// TwinCAT 3 PLC project objectOriented
// ProgramVersion: 3.1.4024.0
// libraries:
//   Tc2_Standard, * (Beckhoff Automation GmbH)
//   Tc2_System, * (Beckhoff Automation GmbH)
//   Tc2_Utilities, * (Beckhoff Automation GmbH)
//   Tc3_Module, * (Beckhoff Automation GmbH)
// project tree:
//   DUTs/ E_EventType.TcDUT, ST_Event.TcDUT
//   / PlcTask.TcTTO
//   POUs/ EventLogger.TcPOU, FB_CsvlPersistentEventStorage.TcPOU, I_PersistentEventStorage.TcIO, MAIN.TcPOU, UpdateEventTimestampWithSystemTime.TcPOU

CONFIGURATION objectOriented
    RESOURCE PLC ON TwinCAT3
        TASK PlcTask(INTERVAL := T#10ms, PRIORITY := 21);
        PROGRAM MAIN WITH PlcTask : MAIN;
    END_RESOURCE
END_CONFIGURATION

// ---- DUTs/E_EventType.TcDUT
{attribute 'qualified_only'}
{attribute 'strict'}
{attribute 'to_string'}
TYPE E_EventType :
(
	Alarm := 0,
	Message := 1
);
END_TYPE

// ---- DUTs/ST_Event.TcDUT
TYPE ST_Event :
STRUCT
	eEventType : E_EventType;
	eEventSeverity : TcEventSeverity;
	nEventIdentity : UDINT;
	sEventText : STRING(255);
	dtTimeStamp : DATE_AND_TIME;
END_STRUCT
END_TYPE

// ---- POUs/I_PersistentEventStorage.TcIO
INTERFACE I_PersistentEventStorage

METHOD StoreEvent
VAR_INPUT
	stEvent : ST_Event;
END_VAR
END_METHOD

END_INTERFACE

// ---- POUs/MAIN.TcPOU
PROGRAM MAIN
VAR
//	UpdateEventTimestam : ST_Event;
	aBoolean : BOOL := FALSE;
		
	eEventType1 : E_EventType := E_EventType.Alarm;
	eEventSeverity1 : TcEventSeverity := TcEventSeverity.Error;
	nEventIdentity1 : UDINT := 42;
	sEventText1 : STRING(255) := 'This is a scary event';
	
	CsvPersistentEventStorage : FB_CsvlPersistentEventStorage;
	EventLogger : EventLogger(CsvPersistentEventStorage); // FB_init call leads to error
END_VAR

//IF NOT aBoolean THEN
//	UpdateEventTimestampWithSystemTime(stEvent := UpdateEventTimestam);
//	aBoolean := TRUE;
//END_IF

IF aBoolean THEN
	EventLogger.AddEvent(eEventType1, eEventSeverity1, nEventIdentity1, sEventText1);
	aBoolean := FALSE;
END_IF

CsvPersistentEventStorage();

END_PROGRAM

// ---- POUs/FB_CsvlPersistentEventStorage.TcPOU
FUNCTION_BLOCK FB_CsvlPersistentEventStorage IMPLEMENTS I_PersistentEventStorage
VAR
	fbFileOpen : FB_FileOpen := (sPathName := 'C:\Events.log', nMode := FOPEN_MODEAPPEND OR FOPEN_MODETEXT);
	fbFilePuts : FB_FilePuts;
	fbFileClose : FB_FileClose;
	eWriteState : (FILE_OPEN_TRIGGER ,FILE_OPEN, WAIT_FOR_EVENT, WRITE_EVENT_TRIGGER, WRITE_EVENT, CLOSE_FILE_TRIGGER, CLOSE_FILE, Error);
	stEventWrittenToFile : ST_Event;
	
	CsvString : T_MaxString;
END_VAR

CASE eWriteState OF
	FILE_OPEN_TRIGGER:
		fbFileOpen(bExecute := TRUE);
		eWriteState := FILE_OPEN;
	
	FILE_OPEN:
		fbFileOpen(bExecute := FALSE);
		IF fbFileOpen.bError THEN
			eWriteState := Error;
		ELSIF NOT fbFileOpen.bBusy AND fbFileOpen.hFile <> 0 THEN
			eWriteState := WAIT_FOR_EVENT;
		END_IF
	
	WAIT_FOR_EVENT:
		//
	WRITE_EVENT_TRIGGER:
		CsvString := CreateCsvString(stEvent := stEventWrittenToFile);
		fbFilePuts(bExecute := TRUE, sLine := CsvString, hFile := fbFileOpen.hFile);
		eWriteState := WRITE_EVENT;
	WRITE_EVENT:
		fbFilePuts(bExecute := FALSE);
		IF fbFilePuts.bError THEN
			eWriteState := Error;
		ELSIF NOT fbFileOpen.bBusy THEN
			eWriteState := CLOSE_FILE_TRIGGER;
		END_IF
	CLOSE_FILE_TRIGGER:
		fbFileClose(bExecute := TRUE, hFile := fbFileOpen.hFile);
		eWriteState := CLOSE_FILE;
	CLOSE_FILE:
		fbFileClose(bExecute := FALSE);
		IF fbFileClose.bError THEN
			eWriteState := Error;
		ELSIF NOT fbFileClose.bBusy THEN
			eWriteState := FILE_OPEN_TRIGGER;
		END_IF
	Error:
	//
	
END_CASE

METHOD PRIVATE CreateCsvString : T_MaxString
VAR_INPUT
	stEvent : REFERENCE TO ST_Event;
END_VAR
VAR
	tempString : T_MaxString;
END_VAR
tempString := TO_STRING(stEvent.eEventType);
tempString := CONCAT(STR1:= tempString, STR2:= ',');
tempString := CONCAT(STR1:= tempString, STR2:= TO_STRING(stEvent.eEventSeverity));
tempString := CONCAT(STR1:= tempString, STR2:= ',');
tempString := CONCAT(STR1:= tempString, STR2:= TO_STRING(stEvent.nEventIdentity));
tempString := CONCAT(STR1:= tempString, STR2:= ',');
tempString := CONCAT(STR1:= tempString, STR2:= stEvent.sEventText);
tempString := CONCAT(STR1:= tempString, STR2:= ',');
tempString := CONCAT(STR1:= tempString, STR2:= TO_STRING(stEvent.dtTimeStamp));
tempString := CONCAT(STR1:= tempString, STR2:= '$n'); // special charecter for next line

CreateCsvString := tempString; // output of method equals its name
END_METHOD

METHOD StoreEvent // error: because Interface just describes the behavior nothing about implementation
VAR_INPUT
	stEvent	: ST_Event;
END_VAR
IF eWriteState = WAIT_FOR_EVENT THEN
	eWriteState := WRITE_EVENT_TRIGGER;
	stEventWrittenToFile := stEvent;
END_IF
END_METHOD

END_FUNCTION_BLOCK

// ---- POUs/EventLogger.TcPOU
FUNCTION_BLOCK EventLogger
VAR
	EventBuffer : ARRAY[1..MAXIMUM_SIZE_OF_EVENT_BUFFER] OF ST_Event;
	CurrentEventBufferIndex : INT := 0;
	_PersistentEventLogger : I_PersistentEventStorage; // (2) store the reference to interface locally in FB
END_VAR
VAR CONSTANT
	MAXIMUM_SIZE_OF_EVENT_BUFFER : INT := 100;
END_VAR

// Returns True if Add was successful and False if the buffer is full
METHOD PUBLIC AddEvent : BOOL
VAR_INPUT
	eEventType : E_EventType;
	eEventSeverity : TcEventSeverity;
	nEventIdentity : UDINT;
	sEventText : STRING(255);
END_VAR
IF NOT IsEventBufferFull() THEN
	CurrentEventBufferIndex := CurrentEventBufferIndex + 1;
	EventBuffer[CurrentEventBufferIndex].eEventType := eEventType;
	EventBuffer[CurrentEventBufferIndex].eEventSeverity := eEventSeverity;
	EventBuffer[CurrentEventBufferIndex].nEventIdentity := nEventIdentity;
	EventBuffer[CurrentEventBufferIndex].sEventText := sEventText;
	UpdateEventTimestampWithSystemTime(stEvent := EventBuffer[CurrentEventBufferIndex]); 
// this function will take a reference to this buffer location and update dtTimastamp of Event
	AddEvent := TRUE;
ELSE
	AddEvent := FALSE;
END_IF
// Here we want to store our Events persistently
_PersistentEventLogger.StoreEvent(stEvent := EventBuffer[CurrentEventBufferIndex]);
END_METHOD

METHOD FB_init : BOOL
VAR_INPUT
	bInitRetains : BOOL; // if TRUE, the retain variables are initialized (warm start / cold start)
	bInCopyCode : BOOL;  // if TRUE, the instance afterwards gets moved into the copy code (online change)
	iPersitentEventStorage : I_PersistentEventStorage; // (1) reference to the interface
END_VAR
_PersistentEventLogger := iPersitentEventStorage; // (3)
END_METHOD

METHOD PRIVATE IsEventBufferFull : BOOL
IF (CurrentEventBufferIndex + 1) > MAXIMUM_SIZE_OF_EVENT_BUFFER THEN
	IsEventBufferFull := TRUE;
ELSE
	IsEventBufferFull := FALSE;
END_IF
END_METHOD

END_FUNCTION_BLOCK

// ---- POUs/UpdateEventTimestampWithSystemTime.TcPOU
FUNCTION UpdateEventTimestampWithSystemTime
VAR_INPUT
	stEvent : REFERENCE TO ST_Event;
END_VAR
VAR
	fbGETSYSTEMTIME : GETSYSTEMTIME;
	stFileName : T_FILETIME;
END_VAR

fbGETSYSTEMTIME(timeLoDW=>stFileName.dwLowDateTime,
 timeHiDW => stFileName.dwHighDateTime);
 
stEvent.dtTimeStamp := FILETIME_TO_DT(fileTime := stFileName);

END_FUNCTION
